// TIA Portal V19 export
FUNCTION "Gros test" : Void   // FC1, LAD
BEGIN

REGION Network 1
   // Voilà un bien gros test...
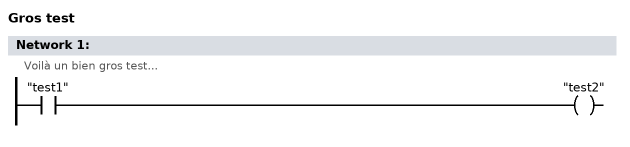
   RUNG wire#powerrail
      Contact( "test1" )
      Coil( "test2" )
   END_RUNG
   // the same network as SCL:
   "test2" := "test1";
END_REGION
END_FUNCTION
